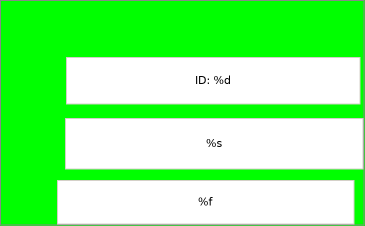
VISUALIZATION Visualization  // 365x226
    Textfield (57,180 297x44), "%f", text variable: PROG_ReadStructure.aReadStruct3.rSinValue
    Textfield (65,118 298x51), "%s", text variable: PROG_ReadStructure.sCzas
    Textfield (66,57 294x47), "ID: %d", text variable: PROG_ReadStructure.aReadStruct3.nID
END_VISUALIZATION

(* stored: Version 1.1.0.1, ProductVersion 3.1.4022.9
   Visu Visualization: Id {4e530394-03e5-4c4e-ab06-4e2dde5972af} *)
